PROGRAM heartbeat_routine
VAR
	opc_heartbeat_error : BOOL;
	heartbeat_ton: TON;
	heartbeat_delay_ton: TON;
	heartbeat_alm_ton: TON;
END_VAR

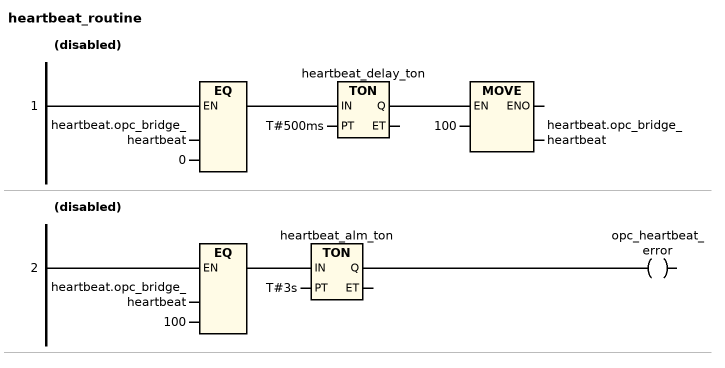
// NETWORK 1 (disabled)
// heartbeat_delay_ton(IN := heartbeat.opc_bridge_heartbeat = 0, PT := T#500ms); // TON
// IF heartbeat_delay_ton.Q THEN heartbeat.opc_bridge_heartbeat := 100; END_IF

// NETWORK 2 (disabled)
// heartbeat_alm_ton(IN := heartbeat.opc_bridge_heartbeat = 100, PT := T#3s); // TON
// opc_heartbeat_error := heartbeat_alm_ton.Q;

END_PROGRAM

(* stored: Version 1.1.0.1, ProductVersion 3.1.4024.15
   POU heartbeat_routine: Id {7cae59a2-e674-46f2-ad40-25d4bb24a618}, SpecialFunc None *)
